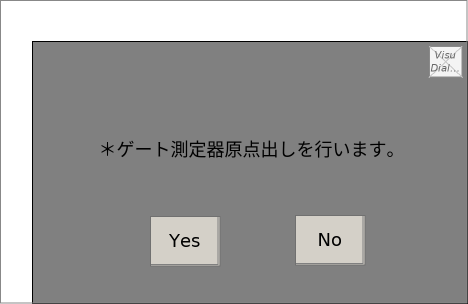
VISUALIZATION d_preset  // 468x304
    Rectangle (32,41 436x263)
    Image (429,46 33x31), image: VisuDialogs.ImagePoolDialogs.Delete
        OnMouseClick: CloseDialog Dialog=d_preset, Result=OK, NumpadKeypadSet=True
    Label (58,105 387x90), "＊ゲート測定器原点出しを行います。"
    Button (150,216 70x50), "Yes"
        tap gvl_visu.flg_btn_gateMeasurementPreset
        OnMouseClick: CloseDialog Dialog=d_preset, Result=OK, NumpadKeypadSet=True
    Button (295,215 70x50), "No"
        OnMouseClick: CloseDialog Dialog=d_preset, Result=OK, NumpadKeypadSet=True
END_VISUALIZATION

(* stored: Version 1.1.0.1, ProductVersion 3.1.4024.12
   Visu d_preset: Id {6cbcc1e3-48c3-43eb-b67a-ce4551a580fa} *)
